// TIA Portal V18 export
ORGANIZATION_BLOCK "Main"   // OB1, LAD, ProgramCycle
TITLE = "Main Program Sweep (Cycle)"
{ S7_Optimized_Access := 'TRUE' }
VERSION : 0.1
// stored: AutoNumber true, IsIECCheckEnabled false, SetENOAutomatically false
   VAR_INPUT
      Initial_Call : Bool;   // Initial call of this OB
      Remanence : Bool;   // =True, if remanent data are available
   END_VAR
   VAR_TEMP   // added for the SCL form of the ladder/FBD networks
      _w1 : Bool;
   END_VAR
BEGIN

REGION Network 1
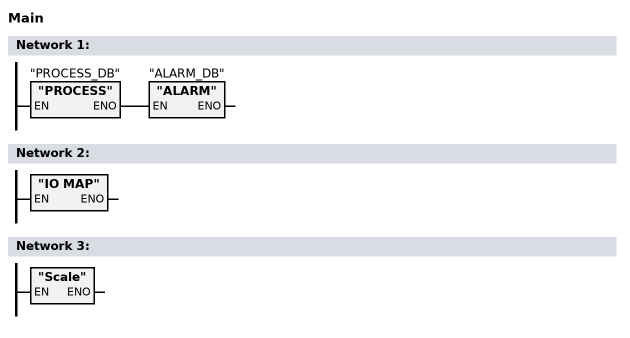
   RUNG wire#powerrail
      "PROCESS_DB"()
      "ALARM_DB"()
   END_RUNG
   // the same network as SCL:
   "PROCESS_DB"(ENO => #_w1);   // "PROCESS"
   IF #_w1 THEN
       "ALARM_DB"();   // "ALARM"
   END_IF;
END_REGION

REGION Network 2
   RUNG wire#powerrail
      "IO MAP"()
   END_RUNG
   // the same network as SCL:
   "IO MAP"();
END_REGION

REGION Network 3
   RUNG wire#powerrail
      "Scale"()
   END_RUNG
   // the same network as SCL:
   "Scale"();
END_REGION
END_ORGANIZATION_BLOCK
